(* PLC project new_app, Dassault Systèmes ControlBuild 2024x Refresh1 *)
(* stored: creationDateTime 2024-04-15T16:43:02-01:00 *)

FUNCTION_BLOCK ffff

END_FUNCTION_BLOCK

PROGRAM new_app.new_app

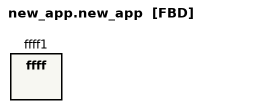
(* FBD diagram, written out as Structured Text *)
ffff1();
END_PROGRAM
